(*			
	RAFALOS
	Rafał Osajda		19.09.2025		TC 4024.66
	Obsługa czasu w systemie
*)
FUNCTION_BLOCK FB_BaseTime IMPLEMENTS ITF_BaseTime
VAR
END_VAR

END_FUNCTION_BLOCK

(* stored: Version 1.1.0.1
   POU FB_BaseTime: Id {aefd6312-b514-007c-3d1e-139902c0f3f6}, SpecialFunc None *)
